# B&R Automation Studio project AGV (part 2)

### libros_topics_typ.c
```c
#include <string.h>
#define EXOS_ASSERT_LOG &logger
#include "exos_log.h"
#include "libros_topics_typ.h"

#define SUCCESS(_format_, ...) exos_log_success(&logger, EXOS_LOG_TYPE_USER, _format_, ##__VA_ARGS__);
#define INFO(_format_, ...) exos_log_info(&logger, EXOS_LOG_TYPE_USER, _format_, ##__VA_ARGS__);
#define VERBOSE(_format_, ...) exos_log_debug(&logger, EXOS_LOG_TYPE_USER + EXOS_LOG_TYPE_VERBOSE, _format_, ##__VA_ARGS__);
#define ERROR(_format_, ...) exos_log_error(&logger, _format_, ##__VA_ARGS__);

static exos_log_handle_t logger;

typedef struct libros_topics_typHandle
{
    libros_topics_typ_t ext_ros_topics_typ_datamodel;
    exos_datamodel_handle_t ros_topics_typ_datamodel;

    exos_dataset_handle_t odemetry_dataset;
    exos_dataset_handle_t twist_dataset;
    exos_dataset_handle_t config_dataset;
} libros_topics_typHandle_t;

static libros_topics_typHandle_t h_ros_topics_typ;

static void libros_topics_typ_datasetEvent(exos_dataset_handle_t *dataset, EXOS_DATASET_EVENT_TYPE event_type, void *info)
{
    switch (event_type)
    {
    case EXOS_DATASET_EVENT_UPDATED:
        VERBOSE("dataset %s updated! latency (us):%i", dataset->name, (exos_datamodel_get_nettime(dataset->datamodel) - dataset->nettime));
        //handle each subscription dataset separately
        if (0 == strcmp(dataset->name, "odemetry"))
        {
            //update the nettime
            h_ros_topics_typ.ext_ros_topics_typ_datamodel.odemetry.nettime = dataset->nettime;

            //trigger the callback if assigned
            if (NULL != h_ros_topics_typ.ext_ros_topics_typ_datamodel.odemetry.on_change)
            {
                h_ros_topics_typ.ext_ros_topics_typ_datamodel.odemetry.on_change();
            }
        }
        break;

    case EXOS_DATASET_EVENT_PUBLISHED:
        break;
    case EXOS_DATASET_EVENT_DELIVERED:
        break;
    case EXOS_DATASET_EVENT_CONNECTION_CHANGED:
        INFO("dataset %s changed state to %s", dataset->name, exos_get_state_string(dataset->connection_state));

        switch (dataset->connection_state)
        {
        case EXOS_STATE_DISCONNECTED:
            break;
        case EXOS_STATE_CONNECTED:
            break;
        case EXOS_STATE_OPERATIONAL:
            break;
        case EXOS_STATE_ABORTED:
            ERROR("dataset %s error %d (%s) occured", dataset->name, dataset->error, exos_get_error_string(dataset->error));
            break;
        }
        break;
    }
}

static void libros_topics_typ_datamodelEvent(exos_datamodel_handle_t *datamodel, const EXOS_DATAMODEL_EVENT_TYPE event_type, void *info)
{
    switch (event_type)
    {
    case EXOS_DATAMODEL_EVENT_CONNECTION_CHANGED:
        INFO("application changed state to %s", exos_get_state_string(datamodel->connection_state));

        h_ros_topics_typ.ext_ros_topics_typ_datamodel.is_connected = false;
        h_ros_topics_typ.ext_ros_topics_typ_datamodel.is_operational = false;
        switch (datamodel->connection_state)
        {
        case EXOS_STATE_DISCONNECTED:
            if (NULL != h_ros_topics_typ.ext_ros_topics_typ_datamodel.on_disconnected)
            {
                h_ros_topics_typ.ext_ros_topics_typ_datamodel.on_disconnected();
            }
            break;
        case EXOS_STATE_CONNECTED:
            h_ros_topics_typ.ext_ros_topics_typ_datamodel.is_connected = true;
            if (NULL != h_ros_topics_typ.ext_ros_topics_typ_datamodel.on_connected)
            {
                h_ros_topics_typ.ext_ros_topics_typ_datamodel.on_connected();
            }
            break;
        case EXOS_STATE_OPERATIONAL:
            h_ros_topics_typ.ext_ros_topics_typ_datamodel.is_connected = true;
            h_ros_topics_typ.ext_ros_topics_typ_datamodel.is_operational = true;
            if (NULL != h_ros_topics_typ.ext_ros_topics_typ_datamodel.on_operational)
            {
                h_ros_topics_typ.ext_ros_topics_typ_datamodel.on_operational();
            }
            SUCCESS("ros_topics_typ operational!");
            break;
        case EXOS_STATE_ABORTED:
            if (NULL != h_ros_topics_typ.ext_ros_topics_typ_datamodel.on_disconnected)
            {
                h_ros_topics_typ.ext_ros_topics_typ_datamodel.on_disconnected();
            }
            ERROR("application error %d (%s) occured", datamodel->error, exos_get_error_string(datamodel->error));
            break;
        }
        break;
    case EXOS_DATAMODEL_EVENT_SYNC_STATE_CHANGED:
        break;

    default:
        break;

    }
}

static void libros_topics_typ_publish_twist_dataset(void)
{
    EXOS_ASSERT_OK(exos_dataset_publish(&h_ros_topics_typ.twist_dataset));
}
static void libros_topics_typ_publish_config_dataset(void)
{
    EXOS_ASSERT_OK(exos_dataset_publish(&h_ros_topics_typ.config_dataset));
}

static void libros_topics_typ_connect(void)
{
    //connect the datamodel
    EXOS_ASSERT_OK(exos_datamodel_connect_ros_topics_typ(&(h_ros_topics_typ.ros_topics_typ_datamodel), libros_topics_typ_datamodelEvent));

    //connect datasets
    EXOS_ASSERT_OK(exos_dataset_connect(&(h_ros_topics_typ.odemetry_dataset), EXOS_DATASET_SUBSCRIBE, libros_topics_typ_datasetEvent));
    EXOS_ASSERT_OK(exos_dataset_connect(&(h_ros_topics_typ.twist_dataset), EXOS_DATASET_PUBLISH, libros_topics_typ_datasetEvent));
    EXOS_ASSERT_OK(exos_dataset_connect(&(h_ros_topics_typ.config_dataset), EXOS_DATASET_PUBLISH, libros_topics_typ_datasetEvent));
}
static void libros_topics_typ_disconnect(void)
{
    h_ros_topics_typ.ext_ros_topics_typ_datamodel.is_connected = false;
    h_ros_topics_typ.ext_ros_topics_typ_datamodel.is_operational = false;

    EXOS_ASSERT_OK(exos_datamodel_disconnect(&(h_ros_topics_typ.ros_topics_typ_datamodel)));
}

static void libros_topics_typ_set_operational(void)
{
    EXOS_ASSERT_OK(exos_datamodel_set_operational(&(h_ros_topics_typ.ros_topics_typ_datamodel)));
}

static void libros_topics_typ_process(void)
{
    EXOS_ASSERT_OK(exos_datamodel_process(&(h_ros_topics_typ.ros_topics_typ_datamodel)));
    exos_log_process(&logger);
}

static void libros_topics_typ_dispose(void)
{
    h_ros_topics_typ.ext_ros_topics_typ_datamodel.is_connected = false;
    h_ros_topics_typ.ext_ros_topics_typ_datamodel.is_operational = false;

    EXOS_ASSERT_OK(exos_datamodel_delete(&(h_ros_topics_typ.ros_topics_typ_datamodel)));
    exos_log_delete(&logger);
}

static int32_t libros_topics_typ_get_nettime(void)
{
    return exos_datamodel_get_nettime(&(h_ros_topics_typ.ros_topics_typ_datamodel));
}

static void libros_topics_typ_log_error(char* log_entry)
{
    exos_log_error(&logger, log_entry);
}

static void libros_topics_typ_log_warning(char* log_entry)
{
    exos_log_warning(&logger, EXOS_LOG_TYPE_USER, log_entry);
}

static void libros_topics_typ_log_success(char* log_entry)
{
    exos_log_success(&logger, EXOS_LOG_TYPE_USER, log_entry);
}

static void libros_topics_typ_log_info(char* log_entry)
{
    exos_log_info(&logger, EXOS_LOG_TYPE_USER, log_entry);
}

static void libros_topics_typ_log_debug(char* log_entry)
{
    exos_log_debug(&logger, EXOS_LOG_TYPE_USER, log_entry);
}

static void libros_topics_typ_log_verbose(char* log_entry)
{
    exos_log_warning(&logger, EXOS_LOG_TYPE_USER + EXOS_LOG_TYPE_VERBOSE, log_entry);
}

libros_topics_typ_t *libros_topics_typ_init(void)
{
    memset(&h_ros_topics_typ, 0, sizeof(h_ros_topics_typ));

    h_ros_topics_typ.ext_ros_topics_typ_datamodel.twist.publish = libros_topics_typ_publish_twist_dataset;
    h_ros_topics_typ.ext_ros_topics_typ_datamodel.config.publish = libros_topics_typ_publish_config_dataset;

    h_ros_topics_typ.ext_ros_topics_typ_datamodel.connect = libros_topics_typ_connect;
    h_ros_topics_typ.ext_ros_topics_typ_datamodel.disconnect = libros_topics_typ_disconnect;
    h_ros_topics_typ.ext_ros_topics_typ_datamodel.process = libros_topics_typ_process;
    h_ros_topics_typ.ext_ros_topics_typ_datamodel.set_operational = libros_topics_typ_set_operational;
    h_ros_topics_typ.ext_ros_topics_typ_datamodel.dispose = libros_topics_typ_dispose;
    h_ros_topics_typ.ext_ros_topics_typ_datamodel.get_nettime = libros_topics_typ_get_nettime;
    h_ros_topics_typ.ext_ros_topics_typ_datamodel.log.error = libros_topics_typ_log_error;
    h_ros_topics_typ.ext_ros_topics_typ_datamodel.log.warning = libros_topics_typ_log_warning;
    h_ros_topics_typ.ext_ros_topics_typ_datamodel.log.success = libros_topics_typ_log_success;
    h_ros_topics_typ.ext_ros_topics_typ_datamodel.log.info = libros_topics_typ_log_info;
    h_ros_topics_typ.ext_ros_topics_typ_datamodel.log.debug = libros_topics_typ_log_debug;
    h_ros_topics_typ.ext_ros_topics_typ_datamodel.log.verbose = libros_topics_typ_log_verbose;

    exos_log_init(&logger, "gros_topics_typ_0");

    SUCCESS("starting gros_topics_typ_0 application..");

    EXOS_ASSERT_OK(exos_datamodel_init(&h_ros_topics_typ.ros_topics_typ_datamodel, "ros_topics_typ_0", "gros_topics_typ_0"));

    //set the user_context to access custom data in the callbacks
    h_ros_topics_typ.ros_topics_typ_datamodel.user_context = NULL; //not used
    h_ros_topics_typ.ros_topics_typ_datamodel.user_tag = 0; //not used

    EXOS_ASSERT_OK(exos_dataset_init(&h_ros_topics_typ.odemetry_dataset, &h_ros_topics_typ.ros_topics_typ_datamodel, "odemetry", &h_ros_topics_typ.ext_ros_topics_typ_datamodel.odemetry.value, sizeof(h_ros_topics_typ.ext_ros_topics_typ_datamodel.odemetry.value)));
    h_ros_topics_typ.odemetry_dataset.user_context = NULL; //not used
    h_ros_topics_typ.odemetry_dataset.user_tag = 0; //not used

    EXOS_ASSERT_OK(exos_dataset_init(&h_ros_topics_typ.twist_dataset, &h_ros_topics_typ.ros_topics_typ_datamodel, "twist", &h_ros_topics_typ.ext_ros_topics_typ_datamodel.twist.value, sizeof(h_ros_topics_typ.ext_ros_topics_typ_datamodel.twist.value)));
    h_ros_topics_typ.twist_dataset.user_context = NULL; //not used
    h_ros_topics_typ.twist_dataset.user_tag = 0; //not used

    EXOS_ASSERT_OK(exos_dataset_init(&h_ros_topics_typ.config_dataset, &h_ros_topics_typ.ros_topics_typ_datamodel, "config", &h_ros_topics_typ.ext_ros_topics_typ_datamodel.config.value, sizeof(h_ros_topics_typ.ext_ros_topics_typ_datamodel.config.value)));
    h_ros_topics_typ.config_dataset.user_context = NULL; //not used
    h_ros_topics_typ.config_dataset.user_tag = 0; //not used

    return &(h_ros_topics_typ.ext_ros_topics_typ_datamodel);
}
```

- libros_topics_typ.i (not shown)

- WaterTank.exospkg - exOS package description (not shown)

### Program Logical/WaterTank/WaterTank_0 (IEC) - WaterTank application

#### WaterTank.var - WaterTank variable declaration
```iecst
VAR
	WaterTank_0 : WaterTank;
	WaterTankCyclic_0 : WaterTankCyclic;
	ExComponentInfo_0 : ExComponentInfo;
	ExDatamodelInfo_0 : ExDatamodelInfo;
	ExDataConnectionInfo_0 : ExDataConnectionInfo;
END_VAR
```

#### WaterTank.st - WaterTank application
```iecst
PROGRAM _INIT

END_PROGRAM

PROGRAM _CYCLIC

    //Auto connect:
    //WaterTankCyclic_0.Enable := ExComponentInfo_0.Operational;
	WaterTankCyclic_0(pWaterTank := ADR(WaterTank_0));

	ExComponentInfo_0(ExTargetLink := ADR(gTarget_0), ExComponentLink := ADR(gWaterTank_0), Enable := TRUE);

	ExDatamodelInfo_0(ExTargetLink := ADR(gTarget_0), Enable := TRUE, InstanceName := 'WaterTank_0');

	ExDataConnectionInfo_0(ExTargetLink := ADR(gTarget_0), Enable := TRUE);

END_PROGRAM

PROGRAM _EXIT

    WaterTankCyclic_0(Enable := FALSE);

END_PROGRAM
```

### Library Logical/WaterTank/WaterTank (ANSIC) - WaterTank exOS library
Depends on: ExData

#### WaterTank.typ - WaterTank datamodel declaration
```iecst
TYPE
	WaterTank : 	STRUCT
		FillValve : VALVE_STATE; (*PUB*)
		EnableHeater : BOOL; (*PUB*)
		HeaterConfig : WaterTankHeaterConfig; (*PUB SUB*)
		Status : WaterTankStatus; (*SUB*)
		StatusDelay : DINT;
		StatusUpdates : UDINT;
	END_STRUCT;
	WaterTankHeaterConfig : 	STRUCT
		MaxTemperature : REAL;
		MaxPower : REAL;
	END_STRUCT;
	WaterTankStatus : 	STRUCT
		LevelHigh : BOOL;
		LevelLow : BOOL;
		FillValveDelay : DINT;
		WaterLevel : DINT;
		Heater : WaterTankHeaterStatus;
	END_STRUCT;
	WaterTankHeaterStatus : 	STRUCT
		WaterTemperature : REAL;
		HeatingActive : BOOL;
	END_STRUCT;
	VALVE_STATE :
		(
		VALVE_CLOSED := 0,
		VALVE_OPEN := 1
		);
END_TYPE
```

#### exos_watertank.h - Generated datamodel header for WaterTank
```c
/*Automatically generated header file from WaterTank.typ*/

#ifndef _EXOS_COMP_WATERTANK_H_
#define _EXOS_COMP_WATERTANK_H_

#include "exos_api.h"

#if defined(_SG4)
#include <WaterTank.h>
#else
#include <stddef.h>
#include <stdint.h>
#include <stdbool.h>

typedef struct WaterTankHeaterStatus
{
    float WaterTemperature;
    bool HeatingActive;

} WaterTankHeaterStatus;

typedef struct WaterTankStatus
{
    bool LevelHigh;
    bool LevelLow;
    int32_t FillValveDelay;
    int32_t WaterLevel;
    struct WaterTankHeaterStatus Heater;

} WaterTankStatus;

typedef struct WaterTankHeaterConfig
{
    float MaxTemperature;
    float MaxPower;

} WaterTankHeaterConfig;

typedef enum VALVE_STATE
{
    VALVE_CLOSED = 0,
    VALVE_OPEN = 1

} VALVE_STATE;

typedef struct WaterTank
{
    VALVE_STATE FillValve; //PUB
    bool EnableHeater; //PUB
    struct WaterTankHeaterConfig HeaterConfig; //PUB SUB
    struct WaterTankStatus Status; //SUB
    int32_t StatusDelay;
    uint32_t StatusUpdates;

} WaterTank;

#endif // _SG4

EXOS_ERROR_CODE exos_datamodel_connect_watertank(exos_datamodel_handle_t *datamodel, exos_datamodel_event_cb datamodel_event_callback);

#endif // _EXOS_COMP_WATERTANK_H_
```

#### exos_watertank.c - Generated datamodel source for WaterTank
```c
/*Automatically generated c file from WaterTank.typ*/

#include "exos_watertank.h"

const char config_watertank[] = "{\"name\":\"struct\",\"attributes\":{\"name\":\"<NAME>\",\"dataType\":\"WaterTank\",\"info\":\"<infoId0>\"},\"children\":[{\"name\":\"enum\",\"attributes\":{\"name\":\"FillValve\",\"dataType\":\"VALVE_STATE\",\"comment\":\"PUB\",\"info\":\"<infoId1>\"},\"children\":[{\"name\":\"value\",\"attributes\":{\"name\":\"VALVE_CLOSED\",\"value\":0}},{\"name\":\"value\",\"attributes\":{\"name\":\"VALVE_OPEN\",\"value\":1}}]},{\"name\":\"variable\",\"attributes\":{\"name\":\"EnableHeater\",\"dataType\":\"BOOL\",\"comment\":\"PUB\",\"info\":\"<infoId2>\"}},{\"name\":\"struct\",\"attributes\":{\"name\":\"HeaterConfig\",\"dataType\":\"WaterTankHeaterConfig\",\"comment\":\"PUB SUB\",\"info\":\"<infoId3>\"},\"children\":[{\"name\":\"variable\",\"attributes\":{\"name\":\"MaxTemperature\",\"dataType\":\"REAL\",\"info\":\"<infoId4>\"}},{\"name\":\"variable\",\"attributes\":{\"name\":\"MaxPower\",\"dataType\":\"REAL\",\"info\":\"<infoId5>\"}}]},{\"name\":\"struct\",\"attributes\":{\"name\":\"Status\",\"dataType\":\"WaterTankStatus\",\"comment\":\"SUB\",\"info\":\"<infoId6>\"},\"children\":[{\"name\":\"variable\",\"attributes\":{\"name\":\"LevelHigh\",\"dataType\":\"BOOL\",\"info\":\"<infoId7>\"}},{\"name\":\"variable\",\"attributes\":{\"name\":\"LevelLow\",\"dataType\":\"BOOL\",\"info\":\"<infoId8>\"}},{\"name\":\"variable\",\"attributes\":{\"name\":\"FillValveDelay\",\"dataType\":\"DINT\",\"info\":\"<infoId9>\"}},{\"name\":\"variable\",\"attributes\":{\"name\":\"WaterLevel\",\"dataType\":\"DINT\",\"info\":\"<infoId10>\"}},{\"name\":\"struct\",\"attributes\":{\"name\":\"Heater\",\"dataType\":\"WaterTankHeaterStatus\",\"info\":\"<infoId11>\"},\"children\":[{\"name\":\"variable\",\"attributes\":{\"name\":\"WaterTemperature\",\"dataType\":\"REAL\",\"info\":\"<infoId12>\"}},{\"name\":\"variable\",\"attributes\":{\"name\":\"HeatingActive\",\"dataType\":\"BOOL\",\"info\":\"<infoId13>\"}}]}]},{\"name\":\"variable\",\"attributes\":{\"name\":\"StatusDelay\",\"dataType\":\"DINT\",\"info\":\"<infoId14>\"}},{\"name\":\"variable\",\"attributes\":{\"name\":\"StatusUpdates\",\"dataType\":\"UDINT\",\"info\":\"<infoId15>\"}}]}";

/*Connect the WaterTank datamodel to the server*/
EXOS_ERROR_CODE exos_datamodel_connect_watertank(exos_datamodel_handle_t *datamodel, exos_datamodel_event_cb datamodel_event_callback)
{
    WaterTank data;
    exos_dataset_info_t datasets[] = {
        {EXOS_DATASET_BROWSE_NAME_INIT,{}},
        {EXOS_DATASET_BROWSE_NAME(FillValve),{}},
        {EXOS_DATASET_BROWSE_NAME(EnableHeater),{}},
        {EXOS_DATASET_BROWSE_NAME(HeaterConfig),{}},
        {EXOS_DATASET_BROWSE_NAME(HeaterConfig.MaxTemperature),{}},
        {EXOS_DATASET_BROWSE_NAME(HeaterConfig.MaxPower),{}},
        {EXOS_DATASET_BROWSE_NAME(Status),{}},
        {EXOS_DATASET_BROWSE_NAME(Status.LevelHigh),{}},
        {EXOS_DATASET_BROWSE_NAME(Status.LevelLow),{}},
        {EXOS_DATASET_BROWSE_NAME(Status.FillValveDelay),{}},
        {EXOS_DATASET_BROWSE_NAME(Status.WaterLevel),{}},
        {EXOS_DATASET_BROWSE_NAME(Status.Heater),{}},
        {EXOS_DATASET_BROWSE_NAME(Status.Heater.WaterTemperature),{}},
        {EXOS_DATASET_BROWSE_NAME(Status.Heater.HeatingActive),{}},
        {EXOS_DATASET_BROWSE_NAME(StatusDelay),{}},
        {EXOS_DATASET_BROWSE_NAME(StatusUpdates),{}}
    };

    exos_datamodel_calc_dataset_info(datasets, sizeof(datasets));

    return exos_datamodel_connect(datamodel, config_watertank, datasets, sizeof(datasets), datamodel_event_callback);
}
```

#### WaterTank.fun - WaterTank function blocks
```iecst
FUNCTION_BLOCK WaterTankCyclic
	VAR_INPUT
		Enable : BOOL;
		Start : BOOL;
		pWaterTank : REFERENCE TO WaterTank;	END_VAR
	VAR_OUTPUT
		Connected : BOOL;
		Operational : BOOL;
		Error : BOOL;
	END_VAR
	VAR
		_Handle : UDINT;
		_Start : BOOL;
		_Enable : BOOL;
	END_VAR
END_FUNCTION_BLOCK
```

#### watertank.c - WaterTank library source
```c
#include <string.h>
#include <stdbool.h>
#include "libwatertank.h"

/* libWaterTank_t datamodel features:

main methods:
    watertank->connect()
    watertank->disconnect()
    watertank->process()
    watertank->set_operational()
    watertank->dispose()
    watertank->get_nettime() : (int32_t) get current nettime

void(void) user callbacks:
    watertank->on_connected
    watertank->on_disconnected
    watertank->on_operational

boolean values:
    watertank->is_connected
    watertank->is_operational

logging methods:
    watertank->log.error(char *)
    watertank->log.warning(char *)
    watertank->log.success(char *)
    watertank->log.info(char *)
    watertank->log.debug(char *)
    watertank->log.verbose(char *)

dataset FillValve:
    watertank->FillValve.publish()
    watertank->FillValve.value : (VALVE_STATE)  actual dataset values

dataset EnableHeater:
    watertank->EnableHeater.publish()
    watertank->EnableHeater.value : (bool)  actual dataset value

dataset HeaterConfig:
    watertank->HeaterConfig.publish()
    watertank->HeaterConfig.on_change : void(void) user callback function
    watertank->HeaterConfig.nettime : (int32_t) nettime @ time of publish
    watertank->HeaterConfig.value : (WaterTankHeaterConfig)  actual dataset values

dataset Status:
    watertank->Status.on_change : void(void) user callback function
    watertank->Status.nettime : (int32_t) nettime @ time of publish
    watertank->Status.value : (WaterTankStatus)  actual dataset values
*/
int snprintf(char *s, size_t n, const char *format, ...);

static libWaterTank_t *watertank;
static struct WaterTankCyclic *cyclic_inst;

static void on_change_heaterconfig(void)
{
    watertank->log.success("dataset config changed, check your new datasets");
    memcpy(&(cyclic_inst->pWaterTank->HeaterConfig), &(watertank->HeaterConfig.value), sizeof(cyclic_inst->pWaterTank->HeaterConfig));
}
static void on_change_status(void)
{
    cyclic_inst->pWaterTank->StatusDelay = watertank->get_nettime() - watertank->Status.nettime;
    cyclic_inst->pWaterTank->StatusUpdates++;

    //check for changes in the received data
    if (watertank->Status.value.LevelHigh > cyclic_inst->pWaterTank->Status.LevelHigh)
    {
        watertank->log.success("Level High reached");
    }
    if (watertank->Status.value.LevelLow > cyclic_inst->pWaterTank->Status.LevelLow)
    {
        watertank->log.success("Level Low reached");
    }
    if (watertank->Status.value.Heater.WaterTemperature != cyclic_inst->pWaterTank->Status.Heater.WaterTemperature)
    {
        char message[256];
        snprintf(message, 256, "Water temperature is now: %f nettime delay: %d us", watertank->Status.value.Heater.WaterTemperature, cyclic_inst->pWaterTank->StatusDelay);
        watertank->log.verbose(message);
    }

    memcpy(&(cyclic_inst->pWaterTank->Status), &(watertank->Status.value), sizeof(cyclic_inst->pWaterTank->Status));
}
_BUR_PUBLIC void WaterTankCyclic(struct WaterTankCyclic *inst)
{
    // check if function block has been created before
    if (cyclic_inst != NULL)
    {
        // return error if more than one function blocks have been created
        if (inst != cyclic_inst)
        {
            inst->Operational = false;
            inst->Connected = false;
            inst->Error = true;
            return;
        }
    }
    cyclic_inst = inst;
    // initialize library
    if ((libWaterTank_t *)inst->_Handle == NULL || (libWaterTank_t *)inst->_Handle != watertank)
    {
        //retrieve the watertank structure
        watertank = libWaterTank_init();

        //setup callbacks
        watertank->HeaterConfig.on_change = on_change_heaterconfig;
        watertank->Status.on_change = on_change_status;

        inst->_Handle = (UDINT)watertank;
    }
    // return error if reference to structure is not set on function block
    if (inst->pWaterTank == NULL)
    {
        inst->Operational = false;
        inst->Connected = false;
        inst->Error = true;
        return;
    }
    if (inst->Enable && !inst->_Enable)
    {
        //connect to the server
        watertank->connect();
    }
    if (!inst->Enable && inst->_Enable)
    {
        //disconnect from server
        cyclic_inst = NULL;
        watertank->disconnect();
    }
    inst->_Enable = inst->Enable;

    if (inst->Start && !inst->_Start && watertank->is_connected)
    {
        watertank->set_operational();
        inst->_Start = inst->Start;
    }
    if (!inst->Start)
    {
        inst->_Start = false;
    }

    //trigger callbacks
    watertank->process();

    if (watertank->is_connected)
    {
        if (memcmp(&(watertank->FillValve.value), &(inst->pWaterTank->FillValve), sizeof(inst->pWaterTank->FillValve)))
        {
            memcpy(&(watertank->FillValve.value), &(inst->pWaterTank->FillValve), sizeof(watertank->FillValve.value));
            watertank->FillValve.publish();
        }

        if (watertank->EnableHeater.value != inst->pWaterTank->EnableHeater)
        {
            watertank->EnableHeater.value = inst->pWaterTank->EnableHeater;
            watertank->EnableHeater.publish();
        }

        if (memcmp(&(watertank->HeaterConfig.value), &(inst->pWaterTank->HeaterConfig), sizeof(inst->pWaterTank->HeaterConfig)))
        {
            memcpy(&(watertank->HeaterConfig.value), &(inst->pWaterTank->HeaterConfig), sizeof(watertank->HeaterConfig.value));
            watertank->HeaterConfig.publish();
        }
    }
    inst->Connected = watertank->is_connected;
    inst->Operational = watertank->is_operational;
}

UINT _EXIT ProgramExit(unsigned long phase)
{
    //shutdown
    watertank->dispose();
    cyclic_inst = NULL;
    return 0;
}
```

#### heapsize.cpp - Dynamic heap configuration
```cpp
unsigned long bur_heap_size = 100000;
```

#### libwatertank.h - WaterTank static library wrapper header
```c
#ifndef _LIBWATERTANK_H_
#define _LIBWATERTANK_H_

#include "exos_watertank.h"

typedef void (*libWaterTank_event_cb)(void);
typedef void (*libWaterTank_method_fn)(void);
typedef int32_t (*libWaterTank_get_nettime_fn)(void);
typedef void (*libWaterTank_log_fn)(char *log_entry);

typedef struct libWaterTankFillValve
{
    libWaterTank_method_fn publish;
    VALVE_STATE value;
} libWaterTankFillValve_t;

typedef struct libWaterTankEnableHeater
{
    libWaterTank_method_fn publish;
    bool value;
} libWaterTankEnableHeater_t;

typedef struct libWaterTankHeaterConfig
{
    libWaterTank_method_fn publish;
    libWaterTank_event_cb on_change;
    int32_t nettime;
    WaterTankHeaterConfig value;
} libWaterTankHeaterConfig_t;

typedef struct libWaterTankStatus
{
    libWaterTank_event_cb on_change;
    int32_t nettime;
    WaterTankStatus value;
} libWaterTankStatus_t;

typedef struct libWaterTank_log
{
    libWaterTank_log_fn error;
    libWaterTank_log_fn warning;
    libWaterTank_log_fn success;
    libWaterTank_log_fn info;
    libWaterTank_log_fn debug;
    libWaterTank_log_fn verbose;
} libWaterTank_log_t;

typedef struct libWaterTank
{
    libWaterTank_method_fn connect;
    libWaterTank_method_fn disconnect;
    libWaterTank_method_fn process;
    libWaterTank_method_fn set_operational;
    libWaterTank_method_fn dispose;
    libWaterTank_get_nettime_fn get_nettime;
    libWaterTank_log_t log;
    libWaterTank_event_cb on_connected;
    libWaterTank_event_cb on_disconnected;
    libWaterTank_event_cb on_operational;
    bool is_connected;
    bool is_operational;
    libWaterTankFillValve_t FillValve;
    libWaterTankEnableHeater_t EnableHeater;
    libWaterTankHeaterConfig_t HeaterConfig;
    libWaterTankStatus_t Status;
} libWaterTank_t;

#ifdef __cplusplus
extern "C" {
#endif
libWaterTank_t *libWaterTank_init(void);
#ifdef __cplusplus
}
#endif
#endif // _LIBWATERTANK_H_
```

#### libwatertank.c - WaterTank static library wrapper source
```c
#include <string.h>
#define EXOS_ASSERT_LOG &logger
#include "exos_log.h"
#include "libwatertank.h"

#define SUCCESS(_format_, ...) exos_log_success(&logger, EXOS_LOG_TYPE_USER, _format_, ##__VA_ARGS__);
#define INFO(_format_, ...) exos_log_info(&logger, EXOS_LOG_TYPE_USER, _format_, ##__VA_ARGS__);
#define VERBOSE(_format_, ...) exos_log_debug(&logger, EXOS_LOG_TYPE_USER + EXOS_LOG_TYPE_VERBOSE, _format_, ##__VA_ARGS__);
#define ERROR(_format_, ...) exos_log_error(&logger, _format_, ##__VA_ARGS__);

static exos_log_handle_t logger;

typedef struct libWaterTankHandle
{
    libWaterTank_t ext_watertank;
    exos_datamodel_handle_t watertank;

    exos_dataset_handle_t fillvalve;
    exos_dataset_handle_t enableheater;
    exos_dataset_handle_t heaterconfig;
    exos_dataset_handle_t status;
} libWaterTankHandle_t;

static libWaterTankHandle_t h_WaterTank;

static void libWaterTank_datasetEvent(exos_dataset_handle_t *dataset, EXOS_DATASET_EVENT_TYPE event_type, void *info)
{
    switch (event_type)
    {
    case EXOS_DATASET_EVENT_UPDATED:
        VERBOSE("dataset %s updated! latency (us):%i", dataset->name, (exos_datamodel_get_nettime(dataset->datamodel) - dataset->nettime));
        //handle each subscription dataset separately
        if (0 == strcmp(dataset->name, "HeaterConfig"))
        {
            //update the nettime
            h_WaterTank.ext_watertank.HeaterConfig.nettime = dataset->nettime;

            //trigger the callback if assigned
            if (NULL != h_WaterTank.ext_watertank.HeaterConfig.on_change)
            {
                h_WaterTank.ext_watertank.HeaterConfig.on_change();
            }
        }
        else if (0 == strcmp(dataset->name, "Status"))
        {
            //update the nettime
            h_WaterTank.ext_watertank.Status.nettime = dataset->nettime;

            //trigger the callback if assigned
            if (NULL != h_WaterTank.ext_watertank.Status.on_change)
            {
                h_WaterTank.ext_watertank.Status.on_change();
            }
        }
        break;

    default:
        break;
    }
}

static void libWaterTank_datamodelEvent(exos_datamodel_handle_t *datamodel, const EXOS_DATAMODEL_EVENT_TYPE event_type, void *info)
{
    switch (event_type)
    {
    case EXOS_DATAMODEL_EVENT_CONNECTION_CHANGED:
        INFO("application changed state to %s", exos_get_state_string(datamodel->connection_state));

        h_WaterTank.ext_watertank.is_connected = false;
        h_WaterTank.ext_watertank.is_operational = false;
        switch (datamodel->connection_state)
        {
        case EXOS_STATE_DISCONNECTED:
            if (NULL != h_WaterTank.ext_watertank.on_disconnected)
            {
                h_WaterTank.ext_watertank.on_disconnected();
            }
            break;
        case EXOS_STATE_CONNECTED:
            h_WaterTank.ext_watertank.is_connected = true;
            if (NULL != h_WaterTank.ext_watertank.on_connected)
            {
                h_WaterTank.ext_watertank.on_connected();
            }
            break;
        case EXOS_STATE_OPERATIONAL:
            h_WaterTank.ext_watertank.is_connected = true;
            h_WaterTank.ext_watertank.is_operational = true;
            if (NULL != h_WaterTank.ext_watertank.on_operational)
            {
                h_WaterTank.ext_watertank.on_operational();
            }
            SUCCESS("WaterTank operational!");
            break;
        case EXOS_STATE_ABORTED:
            if (NULL != h_WaterTank.ext_watertank.on_disconnected)
            {
                h_WaterTank.ext_watertank.on_disconnected();
            }
            ERROR("application error %d (%s) occured", datamodel->error, exos_get_error_string(datamodel->error));
            break;
        }
        break;
    case EXOS_DATAMODEL_EVENT_SYNC_STATE_CHANGED:
        break;

    default:
        break;

    }
}

static void libWaterTank_publish_fillvalve(void)
{
    exos_dataset_publish(&h_WaterTank.fillvalve);
}
static void libWaterTank_publish_enableheater(void)
{
    exos_dataset_publish(&h_WaterTank.enableheater);
}
static void libWaterTank_publish_heaterconfig(void)
{
    exos_dataset_publish(&h_WaterTank.heaterconfig);
}

static void libWaterTank_connect(void)
{
    //connect the datamodel
    EXOS_ASSERT_OK(exos_datamodel_connect_watertank(&(h_WaterTank.watertank), libWaterTank_datamodelEvent));

    //connect datasets
    EXOS_ASSERT_OK(exos_dataset_connect(&(h_WaterTank.fillvalve), EXOS_DATASET_PUBLISH, libWaterTank_datasetEvent));
    EXOS_ASSERT_OK(exos_dataset_connect(&(h_WaterTank.enableheater), EXOS_DATASET_PUBLISH, libWaterTank_datasetEvent));
    EXOS_ASSERT_OK(exos_dataset_connect(&(h_WaterTank.heaterconfig), EXOS_DATASET_PUBLISH + EXOS_DATASET_SUBSCRIBE, libWaterTank_datasetEvent));
    EXOS_ASSERT_OK(exos_dataset_connect(&(h_WaterTank.status), EXOS_DATASET_SUBSCRIBE, libWaterTank_datasetEvent));
}
static void libWaterTank_disconnect(void)
{
    h_WaterTank.ext_watertank.is_connected = false;
    h_WaterTank.ext_watertank.is_operational = false;

    EXOS_ASSERT_OK(exos_datamodel_disconnect(&(h_WaterTank.watertank)));
}

static void libWaterTank_set_operational(void)
{
    EXOS_ASSERT_OK(exos_datamodel_set_operational(&(h_WaterTank.watertank)));
}

static void libWaterTank_process(void)
{
    EXOS_ASSERT_OK(exos_datamodel_process(&(h_WaterTank.watertank)));
    exos_log_process(&logger);
}

static void libWaterTank_dispose(void)
{
    h_WaterTank.ext_watertank.is_connected = false;
    h_WaterTank.ext_watertank.is_operational = false;

    EXOS_ASSERT_OK(exos_datamodel_delete(&(h_WaterTank.watertank)));
    exos_log_delete(&logger);
}

static int32_t libWaterTank_get_nettime(void)
{
    return exos_datamodel_get_nettime(&(h_WaterTank.watertank));
}

static void libWaterTank_log_error(char* log_entry)
{
    exos_log_error(&logger, log_entry);
}

static void libWaterTank_log_warning(char* log_entry)
{
    exos_log_warning(&logger, EXOS_LOG_TYPE_USER, log_entry);
}

static void libWaterTank_log_success(char* log_entry)
{
    exos_log_success(&logger, EXOS_LOG_TYPE_USER, log_entry);
}

static void libWaterTank_log_info(char* log_entry)
{
    exos_log_info(&logger, EXOS_LOG_TYPE_USER, log_entry);
}

static void libWaterTank_log_debug(char* log_entry)
{
    exos_log_debug(&logger, EXOS_LOG_TYPE_USER, log_entry);
}

static void libWaterTank_log_verbose(char* log_entry)
{
    exos_log_warning(&logger, EXOS_LOG_TYPE_USER + EXOS_LOG_TYPE_VERBOSE, log_entry);
}

libWaterTank_t *libWaterTank_init(void)
{
    memset(&h_WaterTank, 0, sizeof(h_WaterTank));

    h_WaterTank.ext_watertank.FillValve.publish = libWaterTank_publish_fillvalve;
    h_WaterTank.ext_watertank.EnableHeater.publish = libWaterTank_publish_enableheater;
    h_WaterTank.ext_watertank.HeaterConfig.publish = libWaterTank_publish_heaterconfig;

    h_WaterTank.ext_watertank.connect = libWaterTank_connect;
    h_WaterTank.ext_watertank.disconnect = libWaterTank_disconnect;
    h_WaterTank.ext_watertank.process = libWaterTank_process;
    h_WaterTank.ext_watertank.set_operational = libWaterTank_set_operational;
    h_WaterTank.ext_watertank.dispose = libWaterTank_dispose;
    h_WaterTank.ext_watertank.get_nettime = libWaterTank_get_nettime;
    h_WaterTank.ext_watertank.log.error = libWaterTank_log_error;
    h_WaterTank.ext_watertank.log.warning = libWaterTank_log_warning;
    h_WaterTank.ext_watertank.log.success = libWaterTank_log_success;
    h_WaterTank.ext_watertank.log.info = libWaterTank_log_info;
    h_WaterTank.ext_watertank.log.debug = libWaterTank_log_debug;
    h_WaterTank.ext_watertank.log.verbose = libWaterTank_log_verbose;

    exos_log_init(&logger, "gWaterTank_0");

    SUCCESS("starting gWaterTank_0 application..");

    EXOS_ASSERT_OK(exos_datamodel_init(&h_WaterTank.watertank, "WaterTank_0", "gWaterTank_0"));

    //set the user_context to access custom data in the callbacks
    h_WaterTank.watertank.user_context = NULL; //not used
    h_WaterTank.watertank.user_tag = 0; //not used

    EXOS_ASSERT_OK(exos_dataset_init(&h_WaterTank.fillvalve, &h_WaterTank.watertank, "FillValve", &h_WaterTank.ext_watertank.FillValve.value, sizeof(h_WaterTank.ext_watertank.FillValve.value)));
    h_WaterTank.fillvalve.user_context = NULL; //not used
    h_WaterTank.fillvalve.user_tag = 0; //not used

    EXOS_ASSERT_OK(exos_dataset_init(&h_WaterTank.enableheater, &h_WaterTank.watertank, "EnableHeater", &h_WaterTank.ext_watertank.EnableHeater.value, sizeof(h_WaterTank.ext_watertank.EnableHeater.value)));
    h_WaterTank.enableheater.user_context = NULL; //not used
    h_WaterTank.enableheater.user_tag = 0; //not used

    EXOS_ASSERT_OK(exos_dataset_init(&h_WaterTank.heaterconfig, &h_WaterTank.watertank, "HeaterConfig", &h_WaterTank.ext_watertank.HeaterConfig.value, sizeof(h_WaterTank.ext_watertank.HeaterConfig.value)));
    h_WaterTank.heaterconfig.user_context = NULL; //not used
    h_WaterTank.heaterconfig.user_tag = 0; //not used

    EXOS_ASSERT_OK(exos_dataset_init(&h_WaterTank.status, &h_WaterTank.watertank, "Status", &h_WaterTank.ext_watertank.Status.value, sizeof(h_WaterTank.ext_watertank.Status.value)));
    h_WaterTank.status.user_context = NULL; //not used
    h_WaterTank.status.user_tag = 0; //not used

    return &(h_WaterTank.ext_watertank);
}
```

### Package Logical/WaterTank/Linux - WaterTank Linux resources

### libwatertank.h - WaterTank static library wrapper header
```c
#ifndef _LIBWATERTANK_H_
#define _LIBWATERTANK_H_

#include "exos_watertank.h"

typedef void (*libWaterTank_event_cb)(void);
typedef void (*libWaterTank_method_fn)(void);
typedef int32_t (*libWaterTank_get_nettime_fn)(void);
typedef void (*libWaterTank_log_fn)(char *log_entry);

typedef struct libWaterTankFillValve
{
    libWaterTank_event_cb on_change;
    int32_t nettime;
    VALVE_STATE value;
} libWaterTankFillValve_t;

typedef struct libWaterTankEnableHeater
{
    libWaterTank_event_cb on_change;
    int32_t nettime;
    bool value;
} libWaterTankEnableHeater_t;

typedef struct libWaterTankHeaterConfig
{
    libWaterTank_method_fn publish;
    libWaterTank_event_cb on_change;
    int32_t nettime;
    WaterTankHeaterConfig value;
} libWaterTankHeaterConfig_t;

typedef struct libWaterTankStatus
{
    libWaterTank_method_fn publish;
    WaterTankStatus value;
} libWaterTankStatus_t;

typedef struct libWaterTank_log
{
    libWaterTank_log_fn error;
    libWaterTank_log_fn warning;
    libWaterTank_log_fn success;
    libWaterTank_log_fn info;
    libWaterTank_log_fn debug;
    libWaterTank_log_fn verbose;
} libWaterTank_log_t;

typedef struct libWaterTank
{
    libWaterTank_method_fn connect;
    libWaterTank_method_fn disconnect;
    libWaterTank_method_fn process;
    libWaterTank_method_fn set_operational;
    libWaterTank_method_fn dispose;
    libWaterTank_get_nettime_fn get_nettime;
    libWaterTank_log_t log;
    libWaterTank_event_cb on_connected;
    libWaterTank_event_cb on_disconnected;
    libWaterTank_event_cb on_operational;
    bool is_connected;
    bool is_operational;
    libWaterTankFillValve_t FillValve;
    libWaterTankEnableHeater_t EnableHeater;
    libWaterTankHeaterConfig_t HeaterConfig;
    libWaterTankStatus_t Status;
} libWaterTank_t;

#ifdef __cplusplus
extern "C" {
#endif
libWaterTank_t *libWaterTank_init(void);
#ifdef __cplusplus
}
#endif
#endif // _LIBWATERTANK_H_
```

### libwatertank.c - WaterTank static library wrapper source
```c
#include <string.h>
#define EXOS_ASSERT_LOG &logger
#include "exos_log.h"
#include "libwatertank.h"

#define SUCCESS(_format_, ...) exos_log_success(&logger, EXOS_LOG_TYPE_USER, _format_, ##__VA_ARGS__);
#define INFO(_format_, ...) exos_log_info(&logger, EXOS_LOG_TYPE_USER, _format_, ##__VA_ARGS__);
#define VERBOSE(_format_, ...) exos_log_debug(&logger, EXOS_LOG_TYPE_USER + EXOS_LOG_TYPE_VERBOSE, _format_, ##__VA_ARGS__);
#define ERROR(_format_, ...) exos_log_error(&logger, _format_, ##__VA_ARGS__);

static exos_log_handle_t logger;

typedef struct libWaterTankHandle
{
    libWaterTank_t ext_watertank;
    exos_datamodel_handle_t watertank;

    exos_dataset_handle_t fillvalve;
    exos_dataset_handle_t enableheater;
    exos_dataset_handle_t heaterconfig;
    exos_dataset_handle_t status;
} libWaterTankHandle_t;

static libWaterTankHandle_t h_WaterTank;

static void libWaterTank_datasetEvent(exos_dataset_handle_t *dataset, EXOS_DATASET_EVENT_TYPE event_type, void *info)
{
    switch (event_type)
    {
    case EXOS_DATASET_EVENT_UPDATED:
        VERBOSE("dataset %s updated! latency (us):%i", dataset->name, (exos_datamodel_get_nettime(dataset->datamodel) - dataset->nettime));
        //handle each subscription dataset separately
        if (0 == strcmp(dataset->name, "FillValve"))
        {
            //update the nettime
            h_WaterTank.ext_watertank.FillValve.nettime = dataset->nettime;

            //trigger the callback if assigned
            if (NULL != h_WaterTank.ext_watertank.FillValve.on_change)
            {
                h_WaterTank.ext_watertank.FillValve.on_change();
            }
        }
        else if (0 == strcmp(dataset->name, "EnableHeater"))
        {
            //update the nettime
            h_WaterTank.ext_watertank.EnableHeater.nettime = dataset->nettime;

            //trigger the callback if assigned
            if (NULL != h_WaterTank.ext_watertank.EnableHeater.on_change)
            {
                h_WaterTank.ext_watertank.EnableHeater.on_change();
            }
        }
        else if (0 == strcmp(dataset->name, "HeaterConfig"))
        {
            //update the nettime
            h_WaterTank.ext_watertank.HeaterConfig.nettime = dataset->nettime;

            //trigger the callback if assigned
            if (NULL != h_WaterTank.ext_watertank.HeaterConfig.on_change)
            {
                h_WaterTank.ext_watertank.HeaterConfig.on_change();
            }
        }
        break;

    default:
        break;
    }
}

static void libWaterTank_datamodelEvent(exos_datamodel_handle_t *datamodel, const EXOS_DATAMODEL_EVENT_TYPE event_type, void *info)
{
    switch (event_type)
    {
    case EXOS_DATAMODEL_EVENT_CONNECTION_CHANGED:
        INFO("application changed state to %s", exos_get_state_string(datamodel->connection_state));

        h_WaterTank.ext_watertank.is_connected = false;
        h_WaterTank.ext_watertank.is_operational = false;
        switch (datamodel->connection_state)
        {
        case EXOS_STATE_DISCONNECTED:
            if (NULL != h_WaterTank.ext_watertank.on_disconnected)
            {
                h_WaterTank.ext_watertank.on_disconnected();
            }
            break;
        case EXOS_STATE_CONNECTED:
            h_WaterTank.ext_watertank.is_connected = true;
            if (NULL != h_WaterTank.ext_watertank.on_connected)
            {
                h_WaterTank.ext_watertank.on_connected();
            }
            break;
        case EXOS_STATE_OPERATIONAL:
            h_WaterTank.ext_watertank.is_connected = true;
            h_WaterTank.ext_watertank.is_operational = true;
            if (NULL != h_WaterTank.ext_watertank.on_operational)
            {
                h_WaterTank.ext_watertank.on_operational();
            }
            SUCCESS("WaterTank operational!");
            break;
        case EXOS_STATE_ABORTED:
            if (NULL != h_WaterTank.ext_watertank.on_disconnected)
            {
                h_WaterTank.ext_watertank.on_disconnected();
            }
            ERROR("application error %d (%s) occured", datamodel->error, exos_get_error_string(datamodel->error));
            break;
        }
        break;
    case EXOS_DATAMODEL_EVENT_SYNC_STATE_CHANGED:
        break;

    default:
        break;

    }
}

static void libWaterTank_publish_heaterconfig(void)
{
    exos_dataset_publish(&h_WaterTank.heaterconfig);
}
static void libWaterTank_publish_status(void)
{
    exos_dataset_publish(&h_WaterTank.status);
}

static void libWaterTank_connect(void)
{
    //connect the datamodel
    EXOS_ASSERT_OK(exos_datamodel_connect_watertank(&(h_WaterTank.watertank), libWaterTank_datamodelEvent));

    //connect datasets
    EXOS_ASSERT_OK(exos_dataset_connect(&(h_WaterTank.fillvalve), EXOS_DATASET_SUBSCRIBE, libWaterTank_datasetEvent));
    EXOS_ASSERT_OK(exos_dataset_connect(&(h_WaterTank.enableheater), EXOS_DATASET_SUBSCRIBE, libWaterTank_datasetEvent));
    EXOS_ASSERT_OK(exos_dataset_connect(&(h_WaterTank.heaterconfig), EXOS_DATASET_PUBLISH + EXOS_DATASET_SUBSCRIBE, libWaterTank_datasetEvent));
    EXOS_ASSERT_OK(exos_dataset_connect(&(h_WaterTank.status), EXOS_DATASET_PUBLISH, libWaterTank_datasetEvent));
}
static void libWaterTank_disconnect(void)
{
    h_WaterTank.ext_watertank.is_connected = false;
    h_WaterTank.ext_watertank.is_operational = false;

    EXOS_ASSERT_OK(exos_datamodel_disconnect(&(h_WaterTank.watertank)));
}

static void libWaterTank_set_operational(void)
{
    EXOS_ASSERT_OK(exos_datamodel_set_operational(&(h_WaterTank.watertank)));
}

static void libWaterTank_process(void)
{
    EXOS_ASSERT_OK(exos_datamodel_process(&(h_WaterTank.watertank)));
    exos_log_process(&logger);
}

static void libWaterTank_dispose(void)
{
    h_WaterTank.ext_watertank.is_connected = false;
    h_WaterTank.ext_watertank.is_operational = false;

    EXOS_ASSERT_OK(exos_datamodel_delete(&(h_WaterTank.watertank)));
    exos_log_delete(&logger);
}

static int32_t libWaterTank_get_nettime(void)
{
    return exos_datamodel_get_nettime(&(h_WaterTank.watertank));
}

static void libWaterTank_log_error(char* log_entry)
{
    exos_log_error(&logger, log_entry);
}

static void libWaterTank_log_warning(char* log_entry)
{
    exos_log_warning(&logger, EXOS_LOG_TYPE_USER, log_entry);
}

static void libWaterTank_log_success(char* log_entry)
{
    exos_log_success(&logger, EXOS_LOG_TYPE_USER, log_entry);
}

static void libWaterTank_log_info(char* log_entry)
{
    exos_log_info(&logger, EXOS_LOG_TYPE_USER, log_entry);
}

static void libWaterTank_log_debug(char* log_entry)
{
    exos_log_debug(&logger, EXOS_LOG_TYPE_USER, log_entry);
}

static void libWaterTank_log_verbose(char* log_entry)
{
    exos_log_warning(&logger, EXOS_LOG_TYPE_USER + EXOS_LOG_TYPE_VERBOSE, log_entry);
}

libWaterTank_t *libWaterTank_init(void)
{
    memset(&h_WaterTank, 0, sizeof(h_WaterTank));

    h_WaterTank.ext_watertank.HeaterConfig.publish = libWaterTank_publish_heaterconfig;
    h_WaterTank.ext_watertank.Status.publish = libWaterTank_publish_status;

    h_WaterTank.ext_watertank.connect = libWaterTank_connect;
    h_WaterTank.ext_watertank.disconnect = libWaterTank_disconnect;
    h_WaterTank.ext_watertank.process = libWaterTank_process;
    h_WaterTank.ext_watertank.set_operational = libWaterTank_set_operational;
    h_WaterTank.ext_watertank.dispose = libWaterTank_dispose;
    h_WaterTank.ext_watertank.get_nettime = libWaterTank_get_nettime;
    h_WaterTank.ext_watertank.log.error = libWaterTank_log_error;
    h_WaterTank.ext_watertank.log.warning = libWaterTank_log_warning;
    h_WaterTank.ext_watertank.log.success = libWaterTank_log_success;
    h_WaterTank.ext_watertank.log.info = libWaterTank_log_info;
    h_WaterTank.ext_watertank.log.debug = libWaterTank_log_debug;
    h_WaterTank.ext_watertank.log.verbose = libWaterTank_log_verbose;

    exos_log_init(&logger, "gWaterTank_0");

    SUCCESS("starting gWaterTank_0 application..");

    EXOS_ASSERT_OK(exos_datamodel_init(&h_WaterTank.watertank, "WaterTank_0", "gWaterTank_0"));

    //set the user_context to access custom data in the callbacks
    h_WaterTank.watertank.user_context = NULL; //not used
    h_WaterTank.watertank.user_tag = 0; //not used

    EXOS_ASSERT_OK(exos_dataset_init(&h_WaterTank.fillvalve, &h_WaterTank.watertank, "FillValve", &h_WaterTank.ext_watertank.FillValve.value, sizeof(h_WaterTank.ext_watertank.FillValve.value)));
    h_WaterTank.fillvalve.user_context = NULL; //not used
    h_WaterTank.fillvalve.user_tag = 0; //not used

    EXOS_ASSERT_OK(exos_dataset_init(&h_WaterTank.enableheater, &h_WaterTank.watertank, "EnableHeater", &h_WaterTank.ext_watertank.EnableHeater.value, sizeof(h_WaterTank.ext_watertank.EnableHeater.value)));
    h_WaterTank.enableheater.user_context = NULL; //not used
    h_WaterTank.enableheater.user_tag = 0; //not used

    EXOS_ASSERT_OK(exos_dataset_init(&h_WaterTank.heaterconfig, &h_WaterTank.watertank, "HeaterConfig", &h_WaterTank.ext_watertank.HeaterConfig.value, sizeof(h_WaterTank.ext_watertank.HeaterConfig.value)));
    h_WaterTank.heaterconfig.user_context = NULL; //not used
    h_WaterTank.heaterconfig.user_tag = 0; //not used

    EXOS_ASSERT_OK(exos_dataset_init(&h_WaterTank.status, &h_WaterTank.watertank, "Status", &h_WaterTank.ext_watertank.Status.value, sizeof(h_WaterTank.ext_watertank.Status.value)));
    h_WaterTank.status.user_context = NULL; //not used
    h_WaterTank.status.user_tag = 0; //not used

    return &(h_WaterTank.ext_watertank);
}
```

- libwatertank.i - SWIG interface file (not shown)

### CMakeLists.txt - CMake build file script
```
cmake_minimum_required(VERSION 3.0)

project(watertank)

set(CMAKE_BUILD_TYPE Debug)
find_package(SWIG REQUIRED)
include(${SWIG_USE_FILE})

# Load Python Libraries
# ---------------------
# a.) use Python 2.7 to avoid version conflicts
find_package(PythonLibs)
# b.) use Python 3 from the distro (same distro used on the target)
# find_package(PythonLibs 3)
# c.) use pyenv to manually install a version matching the Python version on the target distro https://realpython.com/intro-to-pyenv/
# set(PYTHON_INCLUDE_PATH ~/.pyenv/versions/3.5-dev/include/python3.5m)
# set(PYTHON_LIBRARIES ~/.pyenv/versions/3.5-dev/lib/libpython3.5m.so)

include_directories(${PYTHON_INCLUDE_PATH})

include_directories(${CMAKE_CURRENT_SOURCE_DIR})

set(CMAKE_SWIG_FLAGS "")

set(WATERTANK_SOURCES
    libwatertank.c
    libwatertank.i
    exos_watertank.c
    )

set_source_files_properties(${WATERTANK_SOURCES} PROPERTIES CPLUSPLUS ON)

swig_add_module(libWaterTank python ${WATERTANK_SOURCES})
swig_link_libraries(libWaterTank ${PYTHON_LIBRARIES} zmq exos-api)

set(WATERTANK_MODULE_FILES
    build/_libWaterTank.so
    build/libWaterTank.py
    )

install(FILES ${WATERTANK_MODULE_FILES} DESTINATION /home/user/watertank)

set(CPACK_GENERATOR "DEB")
set(CPACK_PACKAGE_NAME exos-comp-watertank)
set(CPACK_PACKAGE_DESCRIPTION_SUMMARY "WaterTank summary")
set(CPACK_PACKAGE_DESCRIPTION "Some description")
set(CPACK_PACKAGE_VENDOR "Your Company")

set(CPACK_PACKAGE_VERSION_MAJOR 1)
set(CPACK_PACKAGE_VERSION_MINOR 0)
set(CPACK_PACKAGE_VERSION_PATCH 0)
set(CPACK_PACKAGE_FILE_NAME exos-comp-watertank_1.0.0_amd64)
set(CPACK_DEBIAN_PACKAGE_MAINTAINER "Your Name")

set(CPACK_DEBIAN_PACKAGE_SHLIBDEPS ON)

include(CPack)
```

- build.sh - build file shell script (not shown)

- watertank.py - Main python script (not shown)

- libWaterTank.py - WaterTank python module (not shown)

- _libWaterTank.so - WaterTank SWIG library (binary file, 536640 bytes)
Listed in the project but not available here: Logical/Global.typ, Logical/Global.var, Logical/Libraries/ROS/Constants.var, Logical/motorCtrl/setupPointers.st, Logical/ros_topics_typ/Linux/exos_ros_topics_typ.h, Logical/ros_topics_typ/Linux/exos_ros_topics_typ.c, Logical/ros_topics_typ/Linux/libros_topics_typ.h, Logical/ros_topics_typ - Copy/motorCtrl/ros_topics_typ.st, Logical/ros_topics_typ - Copy/motorCtrl/setupPointers.st, Logical/ros_topics_typ - Copy/ros_topics/ros_topics_typ.typ, Logical/ros_topics_typ - Copy/ros_topics/exos_ros_topics_typ.h, Logical/ros_topics_typ - Copy/ros_topics/ros_topics.fun, Logical/ros_topics_typ - Copy/ros_topics/ros_topics_typ.c, Logical/ros_topics_typ - Copy/ros_topics/heapsize.cpp, Logical/test/ros_topics_typ/ros_topics_0/ros_topics_typ.var, Logical/WaterTank/Linux/exos_watertank.h, Logical/WaterTank/Linux/exos_watertank.c
